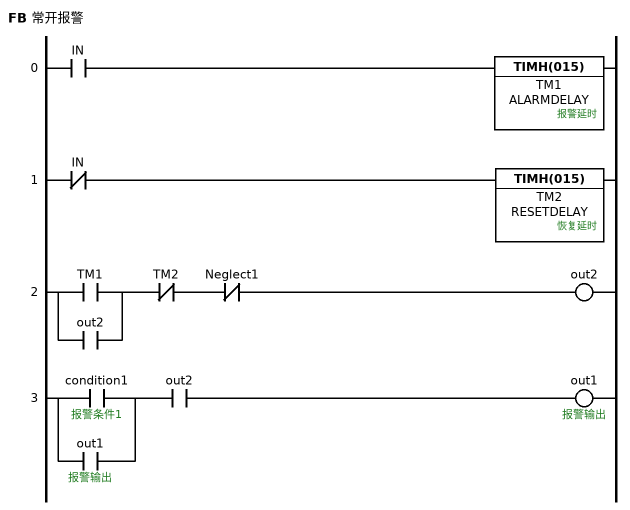
; [picture p24: FB 常开报警, rungs 0-3]
; rung 0
LD IN
TIMH(015) TM1 ALARMDELAY  ; 报警延时
; rung 1
LDNOT IN
TIMH(015) TM2 RESETDELAY  ; 恢复延时
; rung 2
LD TM1
OR out2
ANDNOT TM2
ANDNOT Neglect1
OUT out2
; rung 3
LD condition1  ; 报警条件1
OR out1  ; 报警输出
AND out2
OUT out1  ; 报警输出